// TIA Portal V15.1 export
// export: Created 2024-06-21T08:41:11.8223261Z, ExportSetting WithDefaults, DisplayName Totally Integrated Automation Portal, DisplayVersion V15.1 Update 5, DisplayName TIA Portal Openness, DisplayVersion V15.1 Update 5, DisplayName SINAMICS Startdrive Advanced, DisplayVersion V15.1, DisplayName G130, G150, S120, S150, SINAMICS MV, S210, DisplayVersion V15.1, DisplayName G110M, G120, G120C, G120D, G120P, DisplayVersion V15.1, DisplayName STEP 7 Professional, DisplayVersion V15.1 Update 5, DisplayName STEP 7 Safety, DisplayVersion V15.1, DisplayName WinCC Professional, DisplayVersion V15.1 Update 5, DisplayName SIMATIC Visualization Architect, DisplayVersion V15.1
FUNCTION_BLOCK "LGBShiftRegConv"   // FB6656, FBD
TITLE = LGBShiftRegConv
{ S7_Optimized_Access := 'TRUE' }
VERSION : 0.1
// ============================================================================
// This module is used to shift data between conveyors based on 2 shift sensors and an extra external condition. Data is shifted from previous to actual position.
// The Jobnumber of the previous shift register is cleared after every shift.
// The actual data will be remained untill new date overwrites the old data.
// Alarm generation is based on the Jobnumbers and BodyInPosition.
// Data can be edited by the operator.
// ============================================================================
// stored: AutoNumber false, IsIECCheckEnabled false, IsRetainMemResEnabled false, MemoryReserve 100, SetENOAutomatically False, UDAEnableTagReadback false
   VAR_INPUT
      I_ShiftDet1 { ExternalAccessible := 'False'; ExternalVisible := 'False'; ExternalWritable := 'False'} : Bool := true;   // Shift Detection 1 (Shift cond. 1)
      I_ShiftDet2 { ExternalAccessible := 'False'; ExternalVisible := 'False'; ExternalWritable := 'False'} : Bool := true;   // Shift Detection 2 (Shift cond. 2)
      I_ShiftCond { ExternalAccessible := 'False'; ExternalVisible := 'False'; ExternalWritable := 'False'} : Bool;   // External Shift Condition (Shift cond. 3)
      I_BodyInPosition { ExternalAccessible := 'False'; ExternalVisible := 'False'; ExternalWritable := 'False'} : Bool;   // Body In Position Actual Position
      I_ConvOccupied { ExternalAccessible := 'False'; ExternalVisible := 'False'; ExternalWritable := 'False'} : Bool;   // Conveyor Occupied of Actual Position
      I_ConvRunning { ExternalAccessible := 'False'; ExternalVisible := 'False'; ExternalWritable := 'False'} : Bool;   // Conveyor is running
      I_ShiftReqNext { ExternalAccessible := 'False'; ExternalVisible := 'False'; ExternalWritable := 'False'} : Bool;   // Shift Request of Next Shift Register
      I_EnableAlarm { ExternalAccessible := 'False'; ExternalVisible := 'False'; ExternalWritable := 'False'} : Bool := true;   // Alarm Enable
      I_ResetPB { ExternalAccessible := 'False'; ExternalVisible := 'False'; ExternalWritable := 'False'} : Bool;   // Reset PushButton
      C_MaxOvtShiftReq { ExternalAccessible := 'False'; ExternalVisible := 'False'; ExternalWritable := 'False'} : Time := T#30000ms;   // Maximum Overtime Shift Request
   END_VAR
   VAR_OUTPUT
      O_ShiftRegEmpty { ExternalAccessible := 'False'; ExternalVisible := 'False'; ExternalWritable := 'False'} : Bool;   // Shift Register is Empty
      O_DataOnPosition { ExternalAccessible := 'False'; ExternalVisible := 'False'; ExternalWritable := 'False'} : Bool;   // Data is On Position
      O_ShiftReqActive { ExternalAccessible := 'False'; ExternalVisible := 'False'; ExternalWritable := 'False'} : Bool;   // Shift Request Active
      O_AlarmABCondition { ExternalAccessible := 'False'; ExternalVisible := 'False'; ExternalWritable := 'False'} : Bool;   // Alarm AB condition / Alarm AB Condition
      O_AlarmA { ExternalAccessible := 'False'; ExternalVisible := 'False'; ExternalWritable := 'False'} : Bool;   // Summation Alarm A of roller. / Alarm A
      O_AlarmB { ExternalAccessible := 'False'; ExternalVisible := 'False'; ExternalWritable := 'False'} : Bool;   // Summation Alarm B of roller. / Alarm B
      O_AlarmC { ExternalAccessible := 'False'; ExternalVisible := 'False'; ExternalWritable := 'False'} : Bool;   // Summation Alarm C of roller. / Alarm C
      O_AlarmD { ExternalAccessible := 'False'; ExternalVisible := 'False'; ExternalWritable := 'False'} : Bool;   // Summation Alarm D of roller. / Alarm D
      H_AlarmDWord { ExternalAccessible := 'False'; ExternalVisible := 'False'; ExternalWritable := 'False'} : DWord;   // HMI Animation of the alarms of the roller / Alarm Word
   END_VAR
   VAR_IN_OUT
      H_HMI : "H_HMI";   // Animation
      H_ShiftRegConv : "H_GBShiftRegConv";   // Animation
      IO_ShiftRegConvDataAct : "ShiftRegConvData";   // Data of Actual Position
      IO_ShiftRegConvDataPrev : "ShiftRegConvData";   // Data from Previous Position
   END_VAR
   VAR
      ShiftReqPrevEmptyAlmCond { ExternalAccessible := 'False'; ExternalVisible := 'False'; ExternalWritable := 'False'} : Bool;   // No Jobnumber on Previous Position when Shift is Requested Alarm Condition
      ShiftReqOvtAlmCond { ExternalAccessible := 'False'; ExternalVisible := 'False'; ExternalWritable := 'False'} : Bool;   // Shift Request Overtime Alarm Condition
      BodyInPosActEmptyAlmCond { ExternalAccessible := 'False'; ExternalVisible := 'False'; ExternalWritable := 'False'} : Bool;   // No Jobnumber on Actual Position when Body is In Position and no Shift Request Alarm Condition
      NoBodyInPosActNotEmptyAlmCond { ExternalAccessible := 'False'; ExternalVisible := 'False'; ExternalWritable := 'False'} : Bool;   // Jobnumber on Actual Position when No Body is In Position and no Shift Request Alarm Condition
      AC_ShiftReqPrevEmptyAlm { ExternalAccessible := 'False'; ExternalVisible := 'False'; ExternalWritable := 'False'} : Bool;   // No Jobnumber on Previous Position when Shift is Requested
      AC_ShiftReqOvtAlm { ExternalAccessible := 'False'; ExternalVisible := 'False'; ExternalWritable := 'False'} : Bool;   // Shift Request Overtime
      AC_BodyInPosActEmptyAlm { ExternalAccessible := 'False'; ExternalVisible := 'False'; ExternalWritable := 'False'} : Bool;   // No Jobnumber on Actual Position when Body is In Position and no Shift Request
      AB_NoBodyInPosActNotEmptyAlm { ExternalAccessible := 'False'; ExternalVisible := 'False'; ExternalWritable := 'False'} : Bool;   // Jobnumber on Actual Position when No Body is In Position and no Shift Request
      AD_ChangeDataEnabledWrg { ExternalAccessible := 'False'; ExternalVisible := 'False'; ExternalWritable := 'False'} : Bool;   // Change Data Enabled
      AlarmABCondition { ExternalAccessible := 'False'; ExternalVisible := 'False'; ExternalWritable := 'False'} : Bool;   // Summary of Alarm AB Condition
      AlarmA { ExternalAccessible := 'False'; ExternalVisible := 'False'; ExternalWritable := 'False'} : Bool;   // Summary of Alarm A
      AlarmB { ExternalAccessible := 'False'; ExternalVisible := 'False'; ExternalWritable := 'False'} : Bool;   // Summary of Alarm B
      AlarmC { ExternalAccessible := 'False'; ExternalVisible := 'False'; ExternalWritable := 'False'} : Bool;   // Summary of Alarm C
      AlarmD { ExternalAccessible := 'False'; ExternalVisible := 'False'; ExternalWritable := 'False'} : Bool;   // Summary of Alarm D
      ShiftBegin { ExternalAccessible := 'False'; ExternalVisible := 'False'; ExternalWritable := 'False'} : Bool;   // Begin Actual Shifting
      ShiftBeginTrig { ExternalAccessible := 'False'; ExternalVisible := 'False'; ExternalWritable := 'False'} : Bool;   // Trigger for Begin Actual Shifting
      ShiftRequest { ExternalAccessible := 'False'; ExternalVisible := 'False'; ExternalWritable := 'False'} : Bool;   // Request for Shifting
      ShiftRegEmpty { ExternalAccessible := 'False'; ExternalVisible := 'False'; ExternalWritable := 'False'} : Bool;   // Shift Register Empty
      DataOk { ExternalAccessible := 'False'; ExternalVisible := 'False'; ExternalWritable := 'False'} : Bool;   // Data Ok to Use
      CalculatedGap { ExternalAccessible := 'False'; ExternalVisible := 'False'; ExternalWritable := 'False'} : DWord;   // Gap of data of Actual Shift Register
      ShiftRegConvDataINIT { ExternalAccessible := 'False'; ExternalVisible := 'False'; ExternalWritable := 'False'; S7_SetPoint := 'True'} : "ShiftRegConvData";   // Shift Register Initial Values
      ShiftReqOvt { ExternalAccessible := 'False'; ExternalVisible := 'False'; ExternalWritable := 'False'; S7_SetPoint := 'True'} : "LTimer";   // Shift Request Overtime Timer
   END_VAR
   VAR_TEMP
      HMICmd : Struct   // HMI Commands
         ChangeData : Bool;   // Change Data
         WriteData : Bool;   // Write Data
         DeleteData : Bool;   // Delete Data
         ResetAlarm : Bool;   // Reset Shift Alarm
         BypassWithoutMov : Bool;   // Bypass without movement
         BypassGeneral : Bool;   // Bypass general
         Spare6 : Bool;   // Spare
         Spare7 : Bool;   // Spare
         Spare8 : Bool;   // Spare
         Spare9 : Bool;   // Spare
         Spare10 : Bool;   // Spare
         Spare11 : Bool;   // Spare
         Spare12 : Bool;   // Spare
         Spare13 : Bool;   // Spare
         Spare14 : Bool;   // Spare
         Spare15 : Bool;   // Spare
         Spare16 : Bool;   // Spare
         Spare17 : Bool;   // Spare
         Spare18 : Bool;   // Spare
         Spare19 : Bool;   // Spare
         Spare20 : Bool;   // Spare
         Spare21 : Bool;   // Spare
         Spare22 : Bool;   // Spare
         Spare23 : Bool;   // Spare
         Spare24 : Bool;   // Spare
         Spare25 : Bool;   // Spare
         Spare26 : Bool;   // Spare
         Spare27 : Bool;   // Spare
         Spare28 : Bool;   // Spare
         Spare29 : Bool;   // Spare
         Spare30 : Bool;   // Spare
         Spare31 : Bool;   // Spare
      END_STRUCT;
   END_VAR
   VAR_TEMP   // added for the SCL form of the ladder/FBD networks
      _w1 : Bool;
   END_VAR
BEGIN

REGION Network 1: **** 1 - Inputs **** Extract HMI Commands
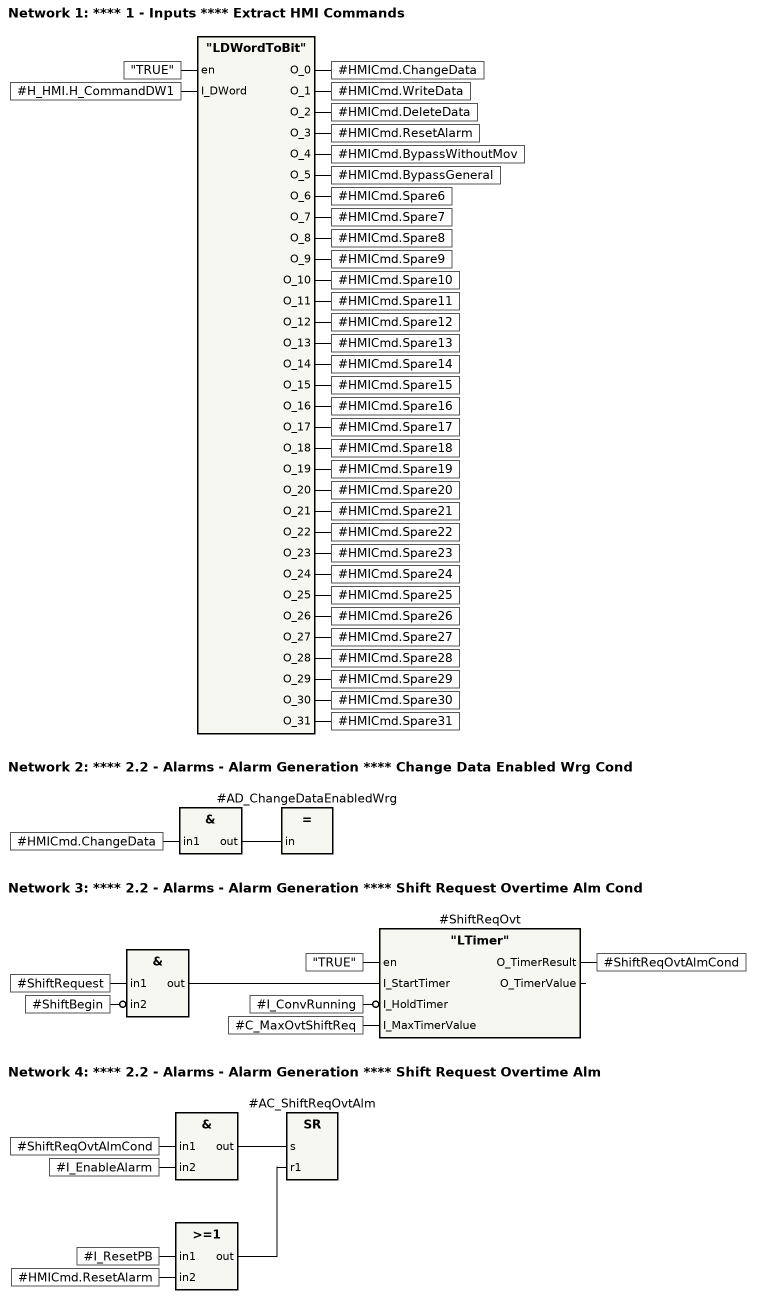
   IF "TRUE" THEN
       "LDWordToBit"(I_DWord := #H_HMI.H_CommandDW1,
                     O_0 => #HMICmd.ChangeData,
                     O_1 => #HMICmd.WriteData,
                     O_2 => #HMICmd.DeleteData,
                     O_3 => #HMICmd.ResetAlarm,
                     O_4 => #HMICmd.BypassWithoutMov,
                     O_5 => #HMICmd.BypassGeneral,
                     O_6 => #HMICmd.Spare6,
                     O_7 => #HMICmd.Spare7,
                     O_8 => #HMICmd.Spare8,
                     O_9 => #HMICmd.Spare9,
                     O_10 => #HMICmd.Spare10,
                     O_11 => #HMICmd.Spare11,
                     O_12 => #HMICmd.Spare12,
                     O_13 => #HMICmd.Spare13,
                     O_14 => #HMICmd.Spare14,
                     O_15 => #HMICmd.Spare15,
                     O_16 => #HMICmd.Spare16,
                     O_17 => #HMICmd.Spare17,
                     O_18 => #HMICmd.Spare18,
                     O_19 => #HMICmd.Spare19,
                     O_20 => #HMICmd.Spare20,
                     O_21 => #HMICmd.Spare21,
                     O_22 => #HMICmd.Spare22,
                     O_23 => #HMICmd.Spare23,
                     O_24 => #HMICmd.Spare24,
                     O_25 => #HMICmd.Spare25,
                     O_26 => #HMICmd.Spare26,
                     O_27 => #HMICmd.Spare27,
                     O_28 => #HMICmd.Spare28,
                     O_29 => #HMICmd.Spare29,
                     O_30 => #HMICmd.Spare30,
                     O_31 => #HMICmd.Spare31);
   END_IF;
END_REGION

REGION Network 2: **** 2.2 - Alarms - Alarm Generation **** Change Data Enabled Wrg Cond
   // Warning Condition
   #AD_ChangeDataEnabledWrg := #HMICmd.ChangeData;
END_REGION

REGION Network 3: **** 2.2 - Alarms - Alarm Generation **** Shift Request Overtime Alm Cond
   // Alarm Condition
   IF "TRUE" THEN
       #ShiftReqOvt(I_StartTimer := #ShiftRequest AND NOT #ShiftBegin,   // "LTimer"
                    I_HoldTimer := NOT #I_ConvRunning,
                    I_MaxTimerValue := #C_MaxOvtShiftReq,
                    O_TimerResult => #ShiftReqOvtAlmCond);
   END_IF;
END_REGION

REGION Network 4: **** 2.2 - Alarms - Alarm Generation **** Shift Request Overtime Alm
   // Alarm C
   IF #ShiftReqOvtAlmCond AND #I_EnableAlarm THEN
       #AC_ShiftReqOvtAlm := TRUE;   // SR flip-flop
   END_IF;
   IF #I_ResetPB OR #HMICmd.ResetAlarm THEN #AC_ShiftReqOvtAlm := FALSE; END_IF;
END_REGION

REGION Network 5: **** 2.2 - Alarms - Alarm Generation **** Body In Position but No Jobnumber Alm Cond
   // Alarm Condition: Actual Position Empty (JobNumber = 0) + Body is In Position (when No Shift Request Active)
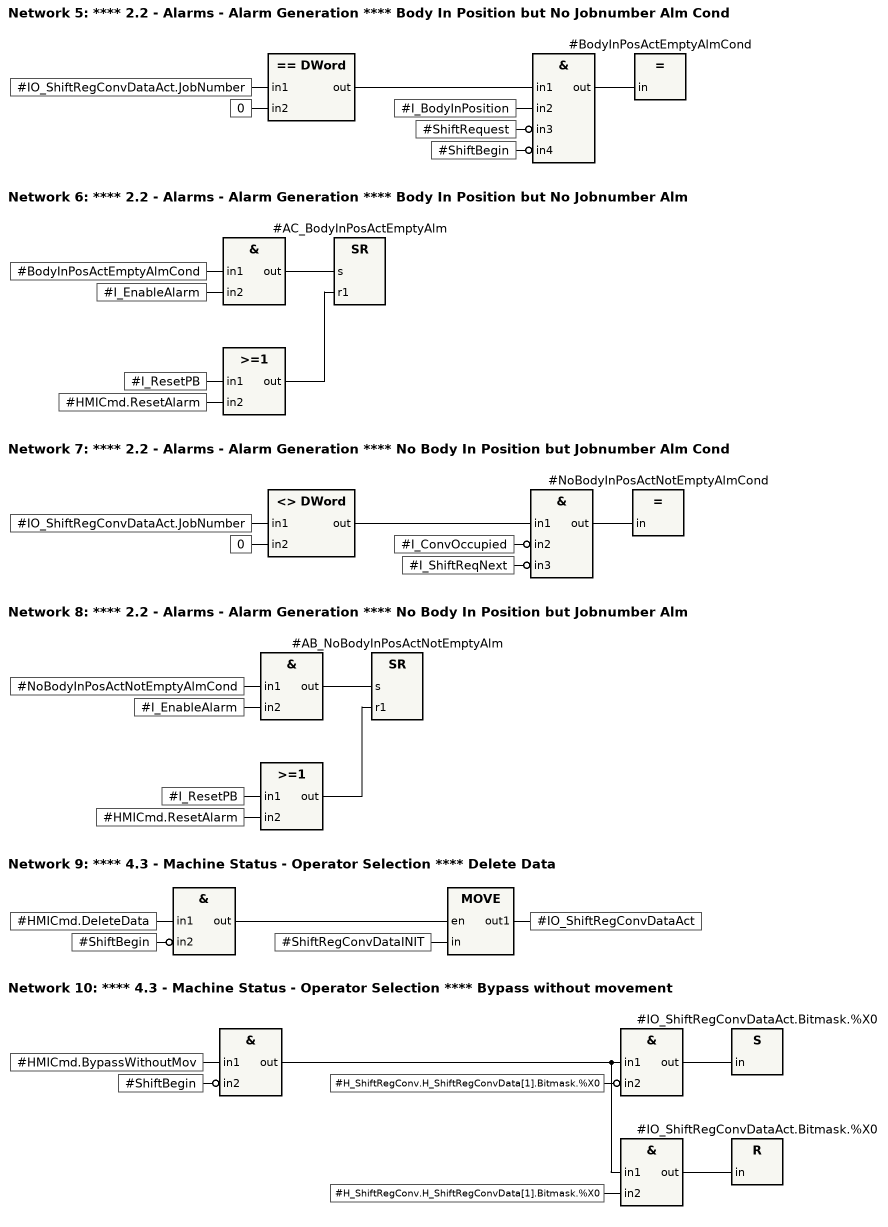
   #BodyInPosActEmptyAlmCond := (#IO_ShiftRegConvDataAct.JobNumber = 0) AND #I_BodyInPosition AND NOT #ShiftRequest AND NOT #ShiftBegin;
END_REGION

REGION Network 6: **** 2.2 - Alarms - Alarm Generation **** Body In Position but No Jobnumber Alm
   // Alarm C
   IF #BodyInPosActEmptyAlmCond AND #I_EnableAlarm THEN
       #AC_BodyInPosActEmptyAlm := TRUE;   // SR flip-flop
   END_IF;
   IF #I_ResetPB OR #HMICmd.ResetAlarm THEN #AC_BodyInPosActEmptyAlm := FALSE; END_IF;
END_REGION

REGION Network 7: **** 2.2 - Alarms - Alarm Generation **** No Body In Position but Jobnumber Alm Cond
   // Alarm Condition: Actual Position Not Empty (JobNumber > 0) + Conveyor Not Occupied (when No Shift Request to Next Position is Active)
   #NoBodyInPosActNotEmptyAlmCond := (#IO_ShiftRegConvDataAct.JobNumber <> 0) AND NOT #I_ConvOccupied AND NOT #I_ShiftReqNext;
END_REGION

REGION Network 8: **** 2.2 - Alarms - Alarm Generation **** No Body In Position but Jobnumber Alm
   // Alarm C
   IF #NoBodyInPosActNotEmptyAlmCond AND #I_EnableAlarm THEN
       #AB_NoBodyInPosActNotEmptyAlm := TRUE;   // SR flip-flop
   END_IF;
   IF #I_ResetPB OR #HMICmd.ResetAlarm THEN #AB_NoBodyInPosActNotEmptyAlm := FALSE; END_IF;
END_REGION

REGION Network 9: **** 4.3 - Machine Status - Operator Selection **** Delete Data
   IF #HMICmd.DeleteData AND NOT #ShiftBegin THEN #IO_ShiftRegConvDataAct := #ShiftRegConvDataINIT; END_IF;
END_REGION

REGION Network 10: **** 4.3 - Machine Status - Operator Selection **** Bypass without movement
   // Write HMI data (edited by operator) to the Shift Register.
   #_w1 := #HMICmd.BypassWithoutMov AND NOT #ShiftBegin;
   IF #_w1 AND NOT #H_ShiftRegConv.H_ShiftRegConvData[1].Bitmask.%X0 THEN
       #IO_ShiftRegConvDataAct.Bitmask.%X0 := TRUE;
   END_IF;
   IF #_w1 AND #H_ShiftRegConv.H_ShiftRegConvData[1].Bitmask.%X0 THEN
       #IO_ShiftRegConvDataAct.Bitmask.%X0 := FALSE;
   END_IF;
END_REGION

REGION Network 11: **** 4.3 - Machine Status - Operator Selection **** Bypass general
   // Write HMI data (edited by operator) to the Shift Register.
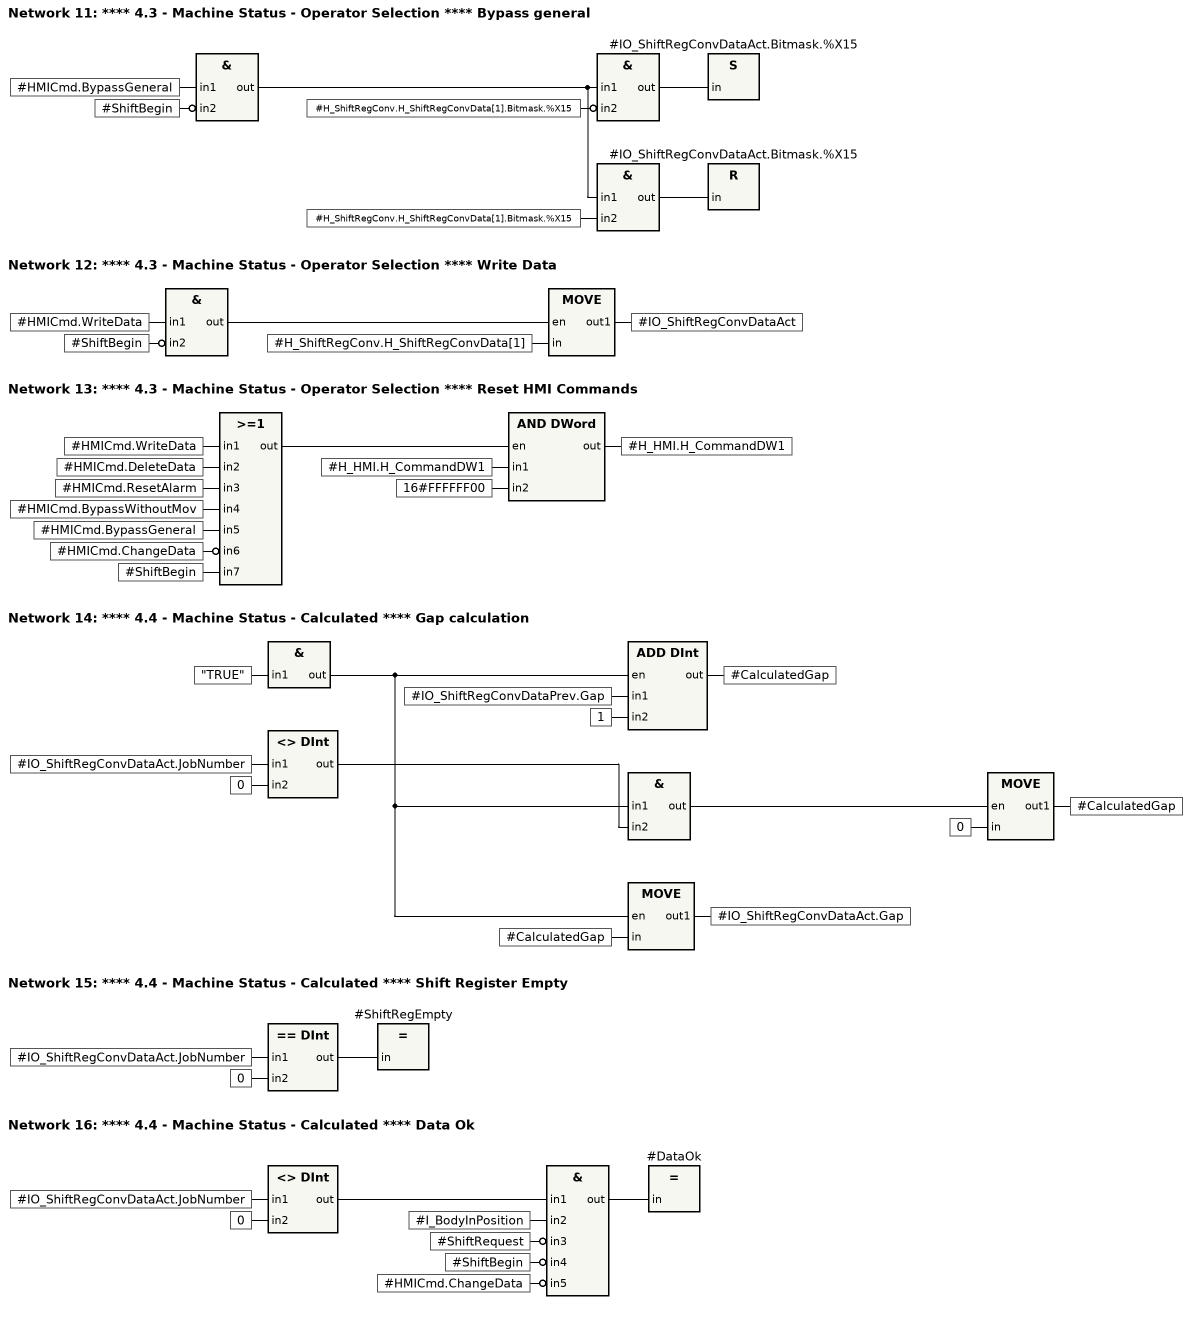
   #_w1 := #HMICmd.BypassGeneral AND NOT #ShiftBegin;
   IF #_w1 AND NOT #H_ShiftRegConv.H_ShiftRegConvData[1].Bitmask.%X15 THEN
       #IO_ShiftRegConvDataAct.Bitmask.%X15 := TRUE;
   END_IF;
   IF #_w1 AND #H_ShiftRegConv.H_ShiftRegConvData[1].Bitmask.%X15 THEN
       #IO_ShiftRegConvDataAct.Bitmask.%X15 := FALSE;
   END_IF;
END_REGION

REGION Network 12: **** 4.3 - Machine Status - Operator Selection **** Write Data
   // Write HMI data (edited by operator) to the Shift Register.
   IF #HMICmd.WriteData AND NOT #ShiftBegin THEN
       #IO_ShiftRegConvDataAct := #H_ShiftRegConv.H_ShiftRegConvData[1];
   END_IF;
END_REGION

REGION Network 13: **** 4.3 - Machine Status - Operator Selection **** Reset HMI Commands
   // Reset HMI Commands when Operator pushes a button or when the Data is Shifted.
   IF #HMICmd.WriteData OR #HMICmd.DeleteData OR #HMICmd.ResetAlarm OR #HMICmd.BypassWithoutMov OR #HMICmd.BypassGeneral OR NOT #HMICmd.ChangeData OR #ShiftBegin THEN
       #H_HMI.H_CommandDW1 := #H_HMI.H_CommandDW1 AND 16#FFFFFF00;
   END_IF;
END_REGION

REGION Network 14: **** 4.4 - Machine Status - Calculated **** Gap calculation
   IF "TRUE" THEN #CalculatedGap := #IO_ShiftRegConvDataPrev.Gap + 1; END_IF;
   IF "TRUE" AND (#IO_ShiftRegConvDataAct.JobNumber <> 0) THEN #CalculatedGap := 0; END_IF;
   IF "TRUE" THEN #IO_ShiftRegConvDataAct.Gap := #CalculatedGap; END_IF;
END_REGION

REGION Network 15: **** 4.4 - Machine Status - Calculated **** Shift Register Empty
   #ShiftRegEmpty := #IO_ShiftRegConvDataAct.JobNumber = 0;
END_REGION

REGION Network 16: **** 4.4 - Machine Status - Calculated **** Data Ok
   // Data is Ok to Use. Body and Associated Data are On Position.
   #DataOk := (#IO_ShiftRegConvDataAct.JobNumber <> 0) AND #I_BodyInPosition AND NOT #ShiftRequest AND NOT #ShiftBegin AND NOT #HMICmd.ChangeData;
END_REGION

REGION Network 17: **** 4.6 - Machine Status - Indication **** Icon Animation
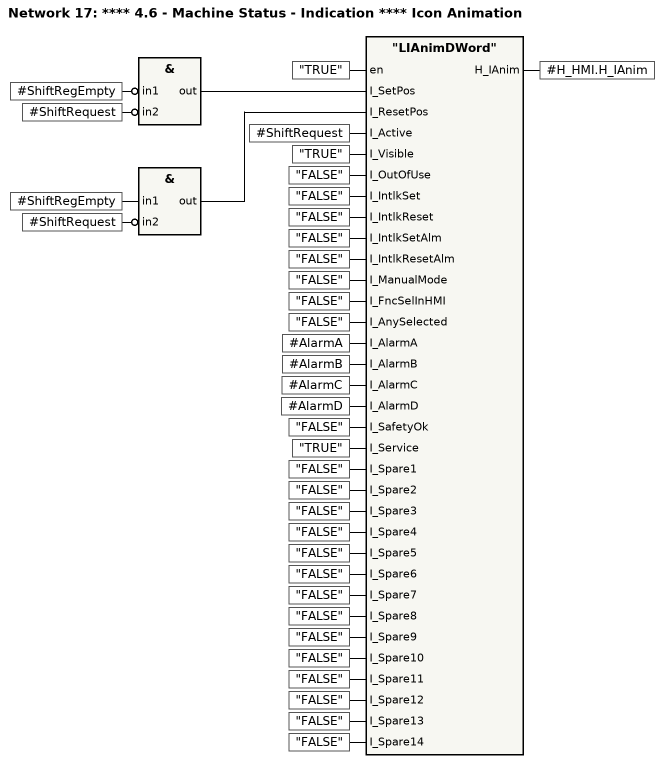
   IF "TRUE" THEN
       "LIAnimDWord"(I_SetPos := NOT #ShiftRegEmpty AND NOT #ShiftRequest,
                     I_ResetPos := #ShiftRegEmpty AND NOT #ShiftRequest,
                     I_Active := #ShiftRequest,
                     I_Visible := "TRUE",
                     I_OutOfUse := "FALSE",
                     I_IntlkSet := "FALSE",
                     I_IntlkReset := "FALSE",
                     I_IntlkSetAlm := "FALSE",
                     I_IntlkResetAlm := "FALSE",
                     I_ManualMode := "FALSE",
                     I_FncSelInHMI := "FALSE",
                     I_AnySelected := "FALSE",
                     I_AlarmA := #AlarmA,
                     I_AlarmB := #AlarmB,
                     I_AlarmC := #AlarmC,
                     I_AlarmD := #AlarmD,
                     I_SafetyOk := "FALSE",
                     I_Service := "TRUE",
                     I_Spare1 := "FALSE",
                     I_Spare2 := "FALSE",
                     I_Spare3 := "FALSE",
                     I_Spare4 := "FALSE",
                     I_Spare5 := "FALSE",
                     I_Spare6 := "FALSE",
                     I_Spare7 := "FALSE",
                     I_Spare8 := "FALSE",
                     I_Spare9 := "FALSE",
                     I_Spare10 := "FALSE",
                     I_Spare11 := "FALSE",
                     I_Spare12 := "FALSE",
                     I_Spare13 := "FALSE",
                     I_Spare14 := "FALSE",
                     H_IAnim => #H_HMI.H_IAnim);
   END_IF;
END_REGION

REGION Network 18: **** 4.6 - Machine Status - Indication **** Animation AnimW1
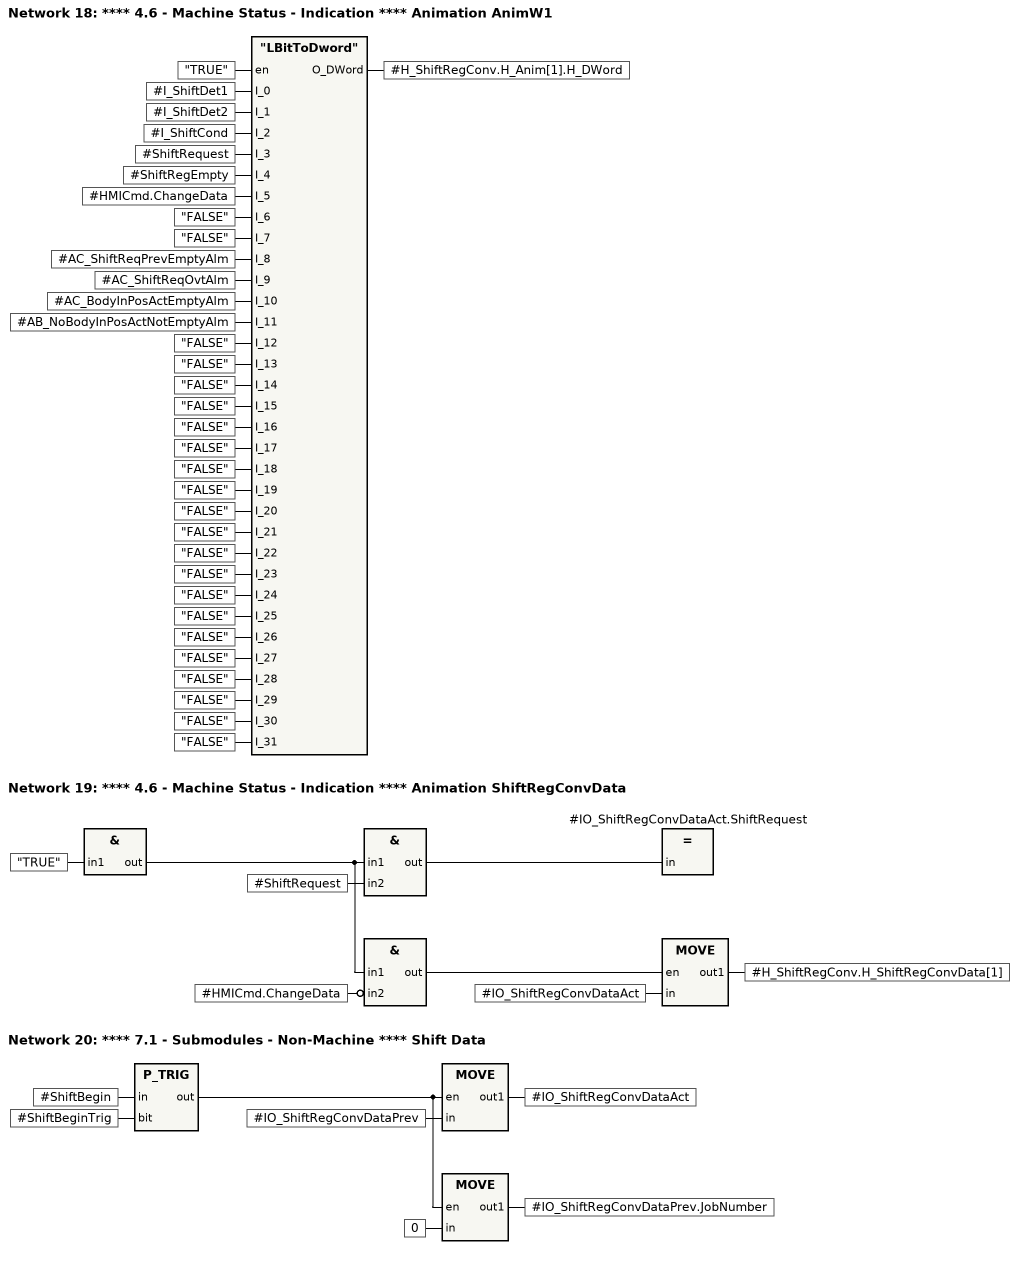
   IF "TRUE" THEN
       "LBitToDword"(I_0 := #I_ShiftDet1,
                     I_1 := #I_ShiftDet2,
                     I_2 := #I_ShiftCond,
                     I_3 := #ShiftRequest,
                     I_4 := #ShiftRegEmpty,
                     I_5 := #HMICmd.ChangeData,
                     I_6 := "FALSE",
                     I_7 := "FALSE",
                     I_8 := #AC_ShiftReqPrevEmptyAlm,
                     I_9 := #AC_ShiftReqOvtAlm,
                     I_10 := #AC_BodyInPosActEmptyAlm,
                     I_11 := #AB_NoBodyInPosActNotEmptyAlm,
                     I_12 := "FALSE",
                     I_13 := "FALSE",
                     I_14 := "FALSE",
                     I_15 := "FALSE",
                     I_16 := "FALSE",
                     I_17 := "FALSE",
                     I_18 := "FALSE",
                     I_19 := "FALSE",
                     I_20 := "FALSE",
                     I_21 := "FALSE",
                     I_22 := "FALSE",
                     I_23 := "FALSE",
                     I_24 := "FALSE",
                     I_25 := "FALSE",
                     I_26 := "FALSE",
                     I_27 := "FALSE",
                     I_28 := "FALSE",
                     I_29 := "FALSE",
                     I_30 := "FALSE",
                     I_31 := "FALSE",
                     O_DWord => #H_ShiftRegConv.H_Anim[1].H_DWord);
   END_IF;
END_REGION

REGION Network 19: **** 4.6 - Machine Status - Indication **** Animation ShiftRegConvData
   #IO_ShiftRegConvDataAct.ShiftRequest := "TRUE" AND #ShiftRequest;
   IF "TRUE" AND NOT #HMICmd.ChangeData THEN
       #H_ShiftRegConv.H_ShiftRegConvData[1] := #IO_ShiftRegConvDataAct;
   END_IF;
END_REGION

REGION Network 20: **** 7.1 - Submodules - Non-Machine **** Shift Data
   #_w1 := #ShiftBegin AND NOT #ShiftBeginTrig;   // rising edge
   #ShiftBeginTrig := #ShiftBegin;
   IF #_w1 THEN
       #IO_ShiftRegConvDataAct := #IO_ShiftRegConvDataPrev;
       #IO_ShiftRegConvDataPrev.JobNumber := 0;
   END_IF;
END_REGION

REGION Network 21: **** 7.2 - Submodules - Command Summary **** Shift Begin
   // Data can be shifted. Set Shift Begin.
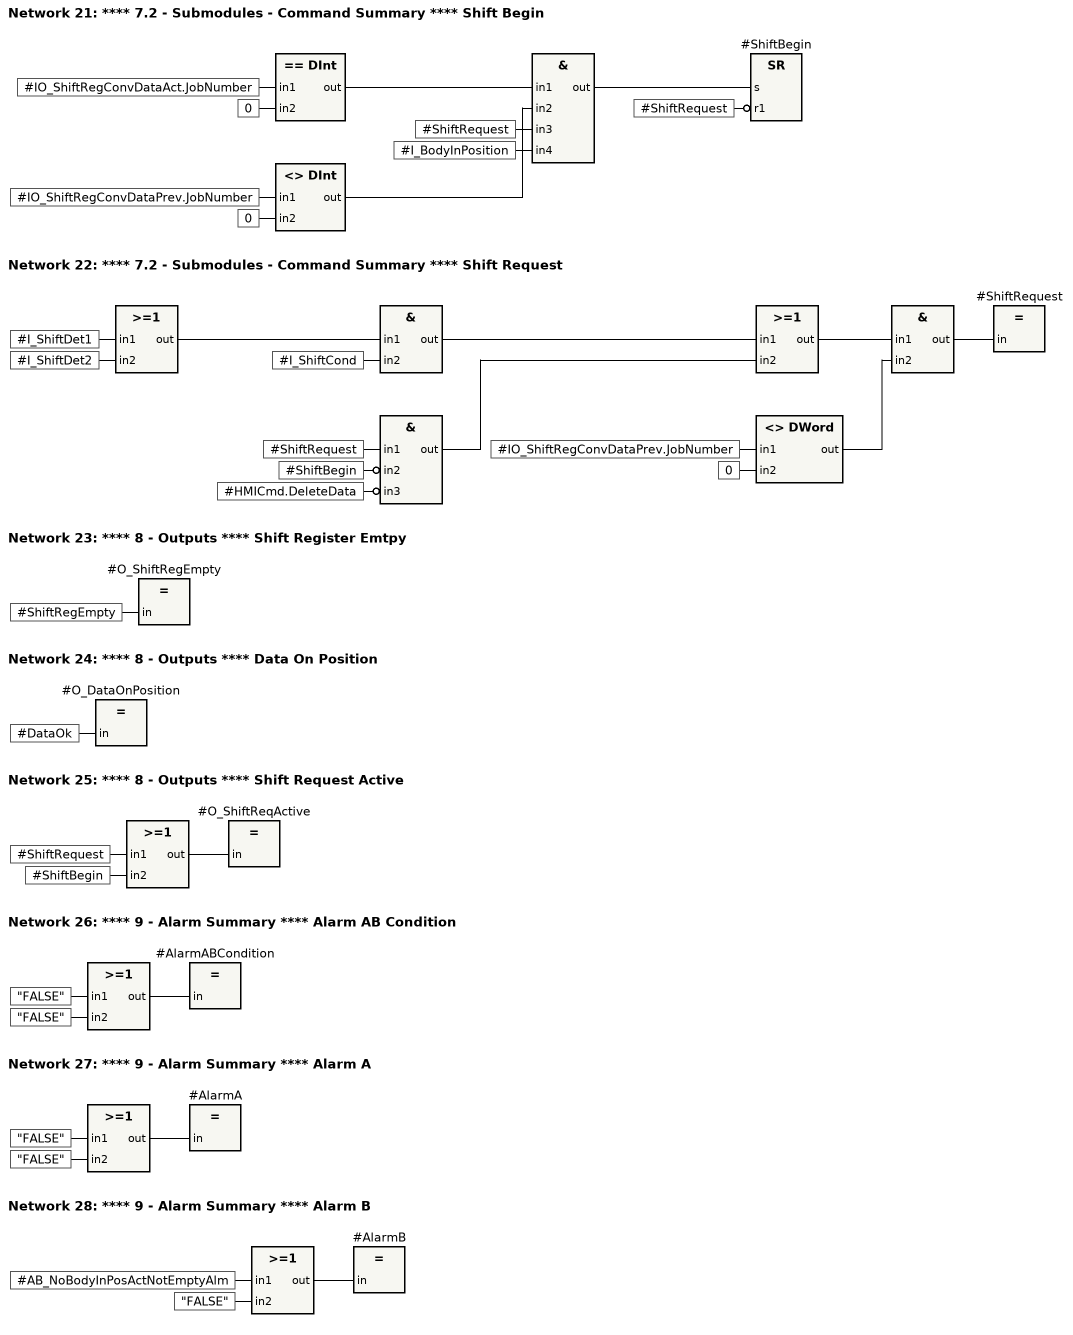
   IF (#IO_ShiftRegConvDataAct.JobNumber = 0) AND (#IO_ShiftRegConvDataPrev.JobNumber <> 0) AND #ShiftRequest AND #I_BodyInPosition THEN
       #ShiftBegin := TRUE;   // SR flip-flop
   END_IF;
   IF NOT #ShiftRequest THEN #ShiftBegin := FALSE; END_IF;
END_REGION

REGION Network 22: **** 7.2 - Submodules - Command Summary **** Shift Request
   // All conditions for shifting are fulfilled. Set Shift Request.
   #ShiftRequest := (((#I_ShiftDet1 OR #I_ShiftDet2) AND #I_ShiftCond) OR (#ShiftRequest AND NOT #ShiftBegin AND NOT #HMICmd.DeleteData)) AND (#IO_ShiftRegConvDataPrev.JobNumber <> 0);
END_REGION

REGION Network 23: **** 8 - Outputs **** Shift Register Emtpy
   #O_ShiftRegEmpty := #ShiftRegEmpty;
END_REGION

REGION Network 24: **** 8 - Outputs **** Data On Position
   #O_DataOnPosition := #DataOk;
END_REGION

REGION Network 25: **** 8 - Outputs **** Shift Request Active
   #O_ShiftReqActive := #ShiftRequest OR #ShiftBegin;
END_REGION

REGION Network 26: **** 9 - Alarm Summary **** Alarm AB Condition
   #AlarmABCondition := "FALSE" OR "FALSE";
END_REGION

REGION Network 27: **** 9 - Alarm Summary **** Alarm A
   // Alarm A
   #AlarmA := "FALSE" OR "FALSE";
END_REGION

REGION Network 28: **** 9 - Alarm Summary **** Alarm B
   // Alarm B
   #AlarmB := #AB_NoBodyInPosActNotEmptyAlm OR "FALSE";
END_REGION

REGION Network 29: **** 9 - Alarm Summary **** Alarm C
   // Alarm C
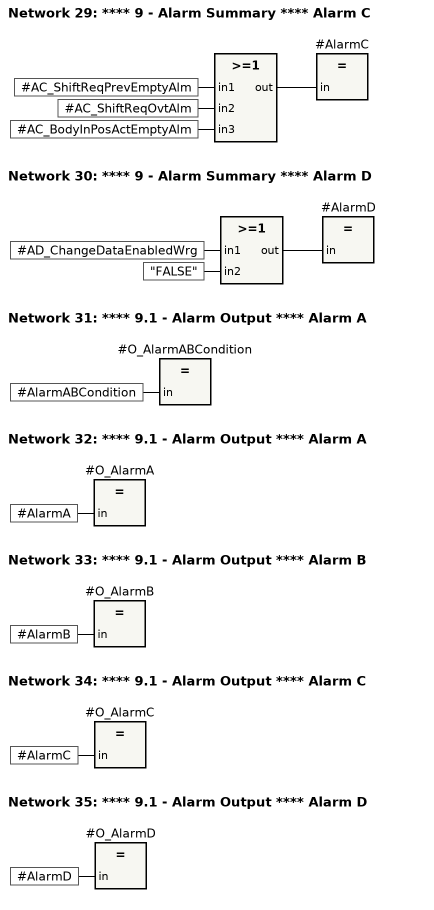
   #AlarmC := #AC_ShiftReqPrevEmptyAlm OR #AC_ShiftReqOvtAlm OR #AC_BodyInPosActEmptyAlm;
END_REGION

REGION Network 30: **** 9 - Alarm Summary **** Alarm D
   // Alarm D
   #AlarmD := #AD_ChangeDataEnabledWrg OR "FALSE";
END_REGION

REGION Network 31: **** 9.1 - Alarm Output **** Alarm A
   // Alarm A
   #O_AlarmABCondition := #AlarmABCondition;
END_REGION

REGION Network 32: **** 9.1 - Alarm Output **** Alarm A
   // Alarm A
   #O_AlarmA := #AlarmA;
END_REGION

REGION Network 33: **** 9.1 - Alarm Output **** Alarm B
   // Alarm B
   #O_AlarmB := #AlarmB;
END_REGION

REGION Network 34: **** 9.1 - Alarm Output **** Alarm C
   // Alarm C
   #O_AlarmC := #AlarmC;
END_REGION

REGION Network 35: **** 9.1 - Alarm Output **** Alarm D
   // Alarm D
   #O_AlarmD := #AlarmD;
END_REGION

REGION Network 36: **** 9.2 - Alarm DWord**** Alarm To DWord
   // Alarm To Word
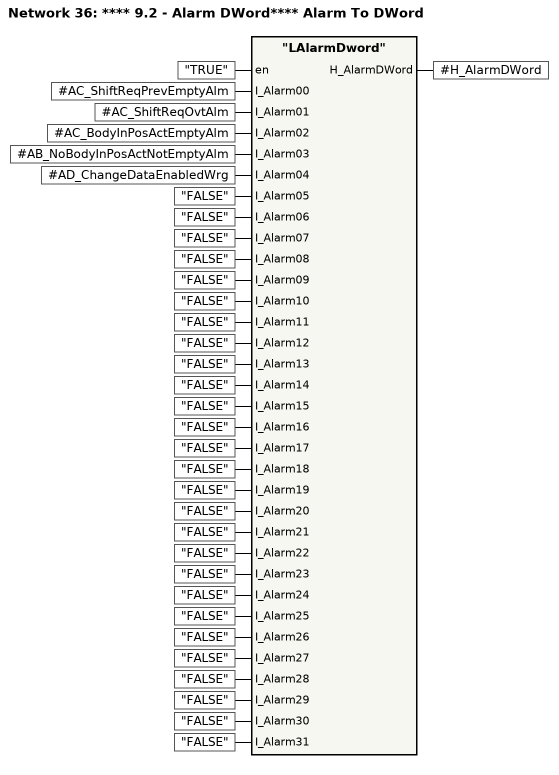
   IF "TRUE" THEN
       "LAlarmDword"(I_Alarm00 := #AC_ShiftReqPrevEmptyAlm,
                     I_Alarm01 := #AC_ShiftReqOvtAlm,
                     I_Alarm02 := #AC_BodyInPosActEmptyAlm,
                     I_Alarm03 := #AB_NoBodyInPosActNotEmptyAlm,
                     I_Alarm04 := #AD_ChangeDataEnabledWrg,
                     I_Alarm05 := "FALSE",
                     I_Alarm06 := "FALSE",
                     I_Alarm07 := "FALSE",
                     I_Alarm08 := "FALSE",
                     I_Alarm09 := "FALSE",
                     I_Alarm10 := "FALSE",
                     I_Alarm11 := "FALSE",
                     I_Alarm12 := "FALSE",
                     I_Alarm13 := "FALSE",
                     I_Alarm14 := "FALSE",
                     I_Alarm15 := "FALSE",
                     I_Alarm16 := "FALSE",
                     I_Alarm17 := "FALSE",
                     I_Alarm18 := "FALSE",
                     I_Alarm19 := "FALSE",
                     I_Alarm20 := "FALSE",
                     I_Alarm21 := "FALSE",
                     I_Alarm22 := "FALSE",
                     I_Alarm23 := "FALSE",
                     I_Alarm24 := "FALSE",
                     I_Alarm25 := "FALSE",
                     I_Alarm26 := "FALSE",
                     I_Alarm27 := "FALSE",
                     I_Alarm28 := "FALSE",
                     I_Alarm29 := "FALSE",
                     I_Alarm30 := "FALSE",
                     I_Alarm31 := "FALSE",
                     H_AlarmDWord => #H_AlarmDWord);
   END_IF;
END_REGION
END_FUNCTION_BLOCK
